TYPE ST_ITC_ATQ :
(**************************************************************************************
 * 	Application		:	BoxControl Framework
 *	Revision		:	$Revision: 404529 $
 *	Revision date	:	$Date: 2018-04-23 08:21:38 +0200 (Mo., 23 Apr 2018) $
 *	Last changed by	:	$Author: b7bolm $
 *	URL				:	$URL: http://almscdc.swisslog.com/repo/SWPD/Development/BoxControlFramework/20_Release/trunk/01_Software/BCF/BCF/JumpStart/20_Product/11_Emu/11_Com/10_Lib/10_Conv/11_ITC/01_DUTs/ST_ITC_ATQ.TcDUT $
 *
 *	Purpose			:	ATQ Structure
 *
 * ------------------------------------------------------------------------------------
 *	Copyright Swisslog [IP AG], Switzerland. All rights reserved.
 * 
 * ------------------------------------------------------------------------------------
 *	
 * 	Revision History: 
 *
 * 	VERSION			DATE			INITIALS			DESCRIPTION
 *	0.1				01.01.2001		swl					Example
 *
 **************************************************************************************)
STRUCT
	Position			: STRING(Conveyor.POSITION_STRINGLENGTH); // SIS position name MM-000-0000-000
	Weight				: DINT; // Weight
	Length				: INT; // length
	Width				: INT; // Width
	Height				: INT; // Height
	LongSideLeading		: BOOL;
	LabelPresent		: INT; // Label present
	Label				: STRING(ConveyorEmulation.LABEL_STRING_LENGTH); // Label
END_STRUCT
END_TYPE

(* stored: Version 1.1.0.1, ProductVersion 3.1.4022.12
   DUT ST_ITC_ATQ: Id {eac1b273-b73f-4f03-a41a-84d3026e355f} *)
